(* PLC project MotionTest1, Higen MCL 1 *)
(* stored: creationDateTime 2012-01-06T15:20:13, modificationDateTime 2026-03-05T12:30:06 *)

PROGRAM main
  VAR
    clock : ULINT;
    Done : BOOL;
    Axis : AXIS_REF;
    switch : MC_Power;
    readtorque : MC_ReadActualTorque;
    Tn : LREAL;
    settorque : MC_TorqueControl;
    my_sim : MC_Sim;
    resettorque : MC_TorqueControl;
    TON0 : TON;
    SR0 : SR;
    SR1 : SR;
  END_VAR

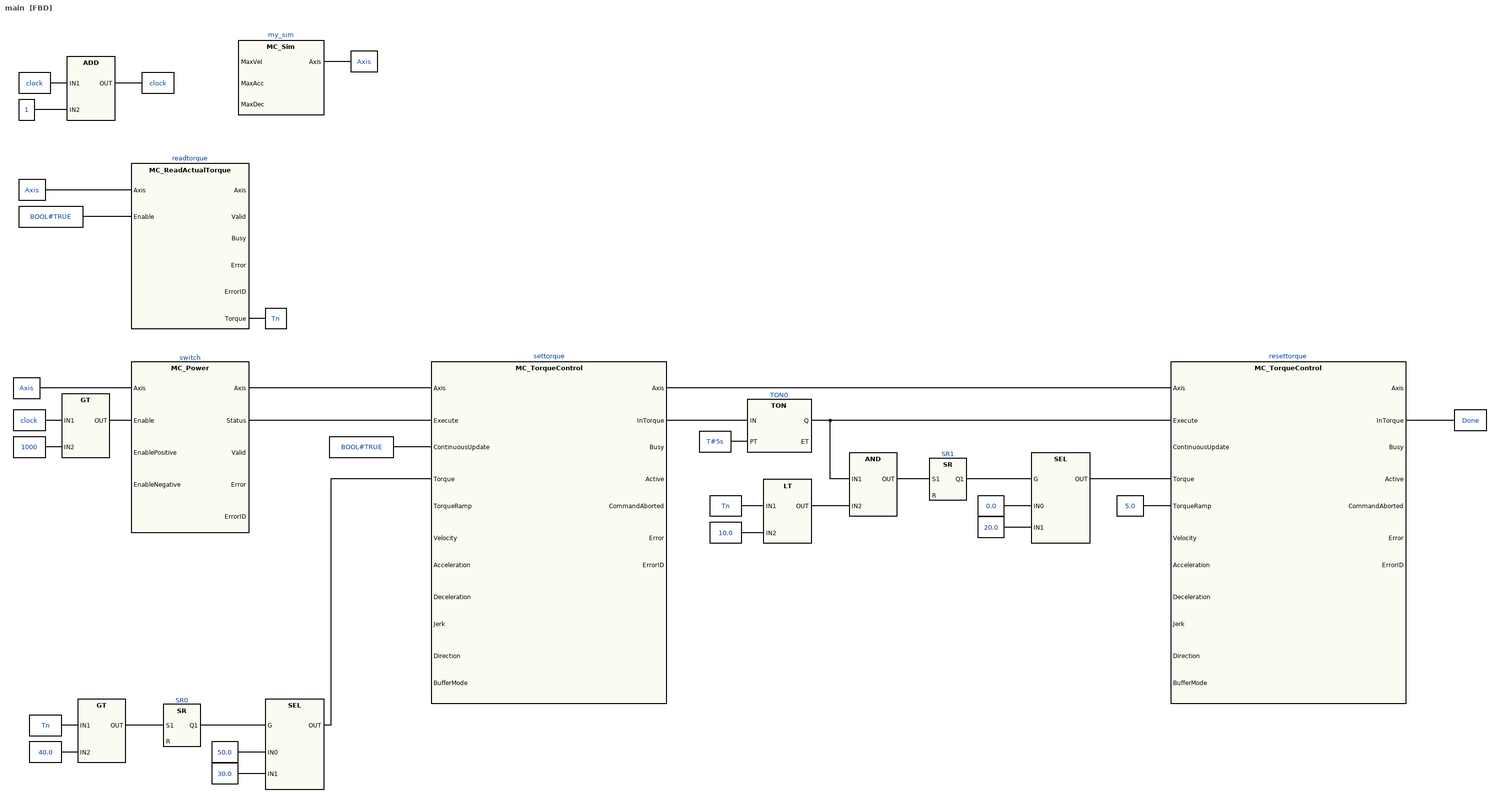
(* FBD diagram, written out as Structured Text *)
clock := clock + 1;
readtorque(Axis := Axis, Enable := BOOL#TRUE);
Tn := readtorque.Torque;
switch(Axis := Axis, Enable := clock > 1000);
SR0(S1 := Tn > 40.0);
settorque(Axis := switch.Axis, Execute := switch.Status, ContinuousUpdate := BOOL#TRUE, Torque := SEL(SR0.Q1, 50.0, 30.0));
TON0(IN := settorque.InTorque, PT := T#5s);
SR1(S1 := TON0.Q AND Tn < 10.0);
resettorque(Axis := settorque.Axis, Execute := TON0.Q, Torque := SEL(SR1.Q1, 0.0, 20.0), TorqueRamp := 5.0);
Done := resettorque.InTorque;
my_sim();
Axis := my_sim.Axis;
END_PROGRAM

CONFIGURATION conf
  RESOURCE res ON PLC
    TASK milisecond(INTERVAL := T#1ms, PRIORITY := 0);
    PROGRAM maininstance WITH milisecond : main;
  END_RESOURCE
END_CONFIGURATION
